// TIA Portal V21 export
VAR_GLOBAL   // PLC tag table "KAllMot"
END_VAR
VAR_GLOBAL CONSTANT   // user constants
   KAllMot_Comunicazione : Int := 1;
   KAllMot_DriveInAllarme : Int := 2;
   KAllMot_Sovracorrente : Int := 3;
   KAllMot_Coppia : Int := 4;
   KAllMot_Termico : Int := 5;
   KAllMot_TimeOutMarcia : Int := 6;
   KAllMot_SezMotoreAperto : Int := 7;
   KAllMot_ScattoTermicoServoventola : Int := 8;
   KAllMot_RichiestaAzzeramento : Int := 9;
   KAllMot_LimiteFisicoPosRaggiunto : Int := 10;
   KAllMot_LimiteFisicoNegRaggiunto : Int := 11;
   KAllMot_MotoreNonInAutoDaHmi : Int := 12;
   KAllMot_MotoreNonInAutoDaPulsLoc : Int := 13;
   KAllMot_FollowingError : Int := 14;
END_VAR
